      movel(p[0.462792, -0.058822, -0.000100, 0.000000, 3.141593, 0.000000],accel_mss,speed_ms,0,blend_radius_m)
      movel(p[0.463472, -0.058210, -0.000100, 0.000000, -3.141593, 0.000000],accel_mss,speed_ms,0,blend_radius_m)
      movel(p[0.463941, -0.057973, -0.000100, 0.000000, -3.141593, 0.000000],accel_mss,speed_ms,0,blend_radius_m)
      movel(p[0.464300, -0.058030, -0.000100, 0.000000, -3.141593, 0.000000],accel_mss,speed_ms,0,0.000)
      movel(p[0.464605, -0.058353, -0.000100, 0.000000, -3.141593, 0.000000],accel_mss,speed_ms,0,0.000)
      movel(p[0.464881, -0.058925, -0.000100, 0.000000, -3.141593, 0.000000],accel_mss,speed_ms,0,blend_radius_m)
      movel(p[0.465128, -0.059615, -0.000100, 0.000000, -3.141593, 0.000000],accel_mss,speed_ms,0,blend_radius_m)
      movel(p[0.465307, -0.060287, -0.000100, 0.000000, -3.141593, 0.000000],accel_mss,speed_ms,0,blend_radius_m)
      movel(p[0.465361, -0.060784, -0.000100, 0.000000, 3.141593, 0.000000],accel_mss,speed_ms,0,0.000)
      movel(p[0.465379, -0.061045, -0.000100, 0.000000, -3.141593, 0.000000],accel_mss,speed_ms,0,0.000)
      movel(p[0.465438, -0.061214, -0.000100, 0.000000, -3.141593, 0.000000],accel_mss,speed_ms,0,0.000)
      movel(p[0.465553, -0.061334, -0.000100, 0.000000, -3.141593, 0.000000],accel_mss,speed_ms,0,0.000)
      movel(p[0.465746, -0.061432, -0.000100, 0.000000, -3.141593, 0.000000],accel_mss,speed_ms,0,0.000)
      movel(p[0.466123, -0.061556, -0.000100, 0.000000, -3.141593, 0.000000],accel_mss,speed_ms,0,0.000)
      movel(p[0.466300, -0.061537, -0.000100, 0.000000, -3.141593, 0.000000],accel_mss,speed_ms,0,0.000)
      movel(p[0.466410, -0.061403, -0.000100, 0.000000, 3.141593, 0.000000],accel_mss,speed_ms,0,0.000)
      movel(p[0.466499, -0.061036, -0.000100, 0.000000, -3.141593, 0.000000],accel_mss,speed_ms,0,0.000)
      movel(p[0.466514, -0.060506, -0.000100, 0.000000, -3.141593, 0.000000],accel_mss,speed_ms,0,blend_radius_m)
      movel(p[0.466371, -0.059685, -0.000100, 0.000000, -3.141593, 0.000000],accel_mss,speed_ms,0,blend_radius_m)
      movel(p[0.466160, -0.058888, -0.000100, 0.000000, 3.141593, 0.000000],accel_mss,speed_ms,0,blend_radius_m)
      movel(p[0.465935, -0.058472, -0.000100, 0.000000, -3.141593, 0.000000],accel_mss,speed_ms,0,0.000)
      movel(p[0.465675, -0.058086, -0.000100, 0.000000, -3.141593, 0.000000],accel_mss,speed_ms,0,0.000)
      movel(p[0.465311, -0.057373, -0.000100, 0.000000, -3.141593, 0.000000],accel_mss,speed_ms,0,blend_radius_m)
      movel(p[0.464973, -0.056642, -0.000100, 0.000000, -3.141593, 0.000000],accel_mss,speed_ms,0,blend_radius_m)
      movel(p[0.464911, -0.056349, -0.000100, 0.000000, 3.141593, 0.000000],accel_mss,speed_ms,0,0.000)
      movel(p[0.464921, -0.056239, -0.000100, 0.000000, -3.141593, 0.000000],accel_mss,speed_ms,0,0.000)
      movel(p[0.464950, -0.056123, -0.000100, 0.000000, -3.141593, 0.000000],accel_mss,speed_ms,0,0.000)
      movel(p[0.464993, -0.056019, -0.000100, 0.000000, -3.141593, 0.000000],accel_mss,speed_ms,0,0.000)
      movel(p[0.465113, -0.055845, -0.000100, 0.000000, -3.141593, 0.000000],accel_mss,speed_ms,0,0.000)
      movel(p[0.465238, -0.055568, -0.000100, 0.000000, -3.141593, 0.000000],accel_mss,speed_ms,0,0.000)
      movel(p[0.465377, -0.055232, -0.000100, 0.000000, 3.141593, 0.000000],accel_mss,speed_ms,0,0.000)
      movel(p[0.465516, -0.054861, -0.000100, 0.000000, -3.141593, 0.000000],accel_mss,speed_ms,0,0.000)
      movel(p[0.465654, -0.054495, -0.000100, 0.000000, -3.141593, 0.000000],accel_mss,speed_ms,0,0.000)
      movel(p[0.465790, -0.054174, -0.000100, 0.000000, -3.141593, 0.000000],accel_mss,speed_ms,0,0.000)
      movel(p[0.465913, -0.053913, -0.000100, 0.000000, -3.141593, 0.000000],accel_mss,speed_ms,0,0.000)
      movel(p[0.466037, -0.053853, -0.000100, 0.000000, -3.141593, 0.000000],accel_mss,speed_ms,0,0.000)
      movel(p[0.466144, -0.053981, -0.000100, 0.000000, -3.141593, 0.000000],accel_mss,speed_ms,0,0.000)
      movel(p[0.466265, -0.054172, -0.000100, 0.000000, -3.141593, 0.000000],accel_mss,speed_ms,0,0.000)
      movel(p[0.466385, -0.054412, -0.000100, 0.000000, -3.141593, 0.000000],accel_mss,speed_ms,0,0.000)
      movel(p[0.466566, -0.054725, -0.000100, 0.000000, -3.141593, 0.000000],accel_mss,speed_ms,0,0.000)
      movel(p[0.466893, -0.055158, -0.000100, 0.000000, 3.141593, 0.000000],accel_mss,speed_ms,0,blend_radius_m)
      movel(p[0.467291, -0.055622, -0.000100, 0.000000, -3.141593, 0.000000],accel_mss,speed_ms,0,blend_radius_m)
      movel(p[0.467706, -0.056051, -0.000100, 0.000000, -3.141593, 0.000000],accel_mss,speed_ms,0,blend_radius_m)
      movel(p[0.468694, -0.056881, -0.000100, 0.000000, -3.141593, 0.000000],accel_mss,speed_ms,0,blend_radius_m)
      movel(p[0.469614, -0.057384, -0.000100, 0.000000, -3.141593, 0.000000],accel_mss,speed_ms,0,blend_radius_m)
      movel(p[0.470598, -0.057620, -0.000100, 0.000000, -3.141593, 0.000000],accel_mss,speed_ms,0,blend_radius_m)
      movel(p[0.471777, -0.057634, -0.000100, 0.000000, -3.141593, 0.000000],accel_mss,speed_ms,0,blend_radius_m)
      movel(p[0.473069, -0.057416, -0.000100, 0.000000, -3.141593, 0.000000],accel_mss,speed_ms,0,blend_radius_m)
      movel(p[0.474031, -0.056974, -0.000100, 0.000000, -3.141593, 0.000000],accel_mss,speed_ms,0,blend_radius_m)
      movel(p[0.474645, -0.056318, -0.000100, 0.000000, -3.141593, 0.000000],accel_mss,speed_ms,0,blend_radius_m)
      movel(p[0.474923, -0.055471, -0.000100, 0.000000, -3.141593, 0.000000],accel_mss,speed_ms,0,blend_radius_m)
      movel(p[0.474946, -0.055083, -0.000100, 0.000000, -3.141593, 0.000000],accel_mss,speed_ms,0,0.000)
      movel(p[0.474919, -0.054836, -0.000100, 0.000000, -3.141593, 0.000000],accel_mss,speed_ms,0,0.000)
      movel(p[0.474836, -0.054649, -0.000100, 0.000000, -3.141593, 0.000000],accel_mss,speed_ms,0,0.000)
      movel(p[0.474680, -0.054470, -0.000100, 0.000000, -3.141593, 0.000000],accel_mss,speed_ms,0,0.000)
      movel(p[0.474476, -0.054300, -0.000100, 0.000000, -3.141593, 0.000000],accel_mss,speed_ms,0,0.000)
      movel(p[0.474370, -0.054271, -0.000100, 0.000000, -3.141593, 0.000000],accel_mss,speed_ms,0,0.000)
      movel(p[0.474268, -0.054324, -0.000100, 0.000000, -3.141593, 0.000000],accel_mss,speed_ms,0,0.000)
      movel(p[0.474075, -0.054545, -0.000100, 0.000000, -3.141593, 0.000000],accel_mss,speed_ms,0,0.000)
      movel(p[0.473962, -0.054704, -0.000100, 0.000000, -3.141593, 0.000000],accel_mss,speed_ms,0,0.000)
      movel(p[0.473898, -0.054846, -0.000100, 0.000000, 3.141593, 0.000000],accel_mss,speed_ms,0,0.000)
      movel(p[0.473884, -0.054962, -0.000100, 0.000000, 3.141593, 0.000000],accel_mss,speed_ms,0,0.000)
      movel(p[0.473977, -0.055623, -0.000100, 0.000000, -3.141593, 0.000000],accel_mss,speed_ms,0,blend_radius_m)
      movel(p[0.473290, -0.056328, -0.000100, 0.000000, -3.141593, 0.000000],accel_mss,speed_ms,0,blend_radius_m)
      movel(p[0.472150, -0.056906, -0.000100, 0.000000, -3.141593, 0.000000],accel_mss,speed_ms,0,blend_radius_m)
      movel(p[0.470974, -0.057097, -0.000100, 0.000000, 3.141593, 0.000000],accel_mss,speed_ms,0,blend_radius_m)
      movel(p[0.470387, -0.057058, -0.000100, 0.000000, -3.141593, 0.000000],accel_mss,speed_ms,0,blend_radius_m)
      movel(p[0.469879, -0.056952, -0.000100, 0.000000, -3.141593, 0.000000],accel_mss,speed_ms,0,blend_radius_m)
      movel(p[0.469515, -0.056804, -0.000100, 0.000000, -3.141593, 0.000000],accel_mss,speed_ms,0,0.000)
      movel(p[0.469411, -0.056632, -0.000100, 0.000000, -3.141593, 0.000000],accel_mss,speed_ms,0,0.000)
      movel(p[0.469349, -0.056523, -0.000100, 0.000000, -3.141593, 0.000000],accel_mss,speed_ms,0,0.000)
      movel(p[0.469199, -0.056478, -0.000100, 0.000000, -3.141593, 0.000000],accel_mss,speed_ms,0,0.000)
      movel(p[0.468853, -0.056330, -0.000100, 0.000000, -3.141593, 0.000000],accel_mss,speed_ms,0,0.000)
      movel(p[0.467795, -0.055190, -0.000100, 0.000000, -3.141593, 0.000000],accel_mss,speed_ms,0,blend_radius_m)
      movel(p[0.466811, -0.054046, -0.000100, 0.000000, 3.141593, 0.000000],accel_mss,speed_ms,0,blend_radius_m)
      movel(p[0.466321, -0.053296, -0.000100, 0.000000, -3.141593, 0.000000],accel_mss,speed_ms,0,blend_radius_m)
      movel(p[0.466173, -0.052959, -0.000100, 0.000000, -3.141593, 0.000000],accel_mss,speed_ms,0,0.000)
      movel(p[0.466058, -0.052599, -0.000100, 0.000000, -3.141593, 0.000000],accel_mss,speed_ms,0,0.000)
      movel(p[0.465985, -0.052243, -0.000100, 0.000000, 3.141593, 0.000000],accel_mss,speed_ms,0,0.000)
      movel(p[0.465961, -0.051920, -0.000100, 0.000000, -3.141593, 0.000000],accel_mss,speed_ms,0,0.000)
      movel(p[0.465948, -0.051608, -0.000100, 0.000000, -3.141593, 0.000000],accel_mss,speed_ms,0,0.000)
      movel(p[0.465908, -0.051219, -0.000100, 0.000000, 3.141593, 0.000000],accel_mss,speed_ms,0,0.000)
      movel(p[0.465850, -0.050819, -0.000100, 0.000000, 3.141593, 0.000000],accel_mss,speed_ms,0,0.000)
      movel(p[0.465781, -0.050472, -0.000100, 0.000000, -3.141593, 0.000000],accel_mss,speed_ms,0,0.000)
      movel(p[0.465685, -0.050012, -0.000100, 0.000000, -3.141593, 0.000000],accel_mss,speed_ms,0,0.000)
      movel(p[0.465675, -0.049785, -0.000100, 0.000000, -3.141593, 0.000000],accel_mss,speed_ms,0,0.000)
      movel(p[0.465734, -0.049633, -0.000100, 0.000000, -3.141593, 0.000000],accel_mss,speed_ms,0,0.000)
      movel(p[0.465878, -0.049490, -0.000100, 0.000000, 3.141593, 0.000000],accel_mss,speed_ms,0,0.000)
      movel(p[0.465992, -0.049418, -0.000100, 0.000000, -3.141593, 0.000000],accel_mss,speed_ms,0,0.000)
      movel(p[0.466107, -0.049368, -0.000100, 0.000000, -3.141593, 0.000000],accel_mss,speed_ms,0,0.000)
      movel(p[0.466205, -0.049344, -0.000100, 0.000000, -3.141593, 0.000000],accel_mss,speed_ms,0,0.000)
      movel(p[0.466337, -0.049355, -0.000100, 0.000000, -3.141593, 0.000000],accel_mss,speed_ms,0,0.000)
      movel(p[0.466507, -0.049227, -0.000100, 0.000000, -3.141593, 0.000000],accel_mss,speed_ms,0,0.000)
      movel(p[0.466710, -0.049045, -0.000100, 0.000000, -3.141593, 0.000000],accel_mss,speed_ms,0,0.000)
      movel(p[0.466929, -0.048816, -0.000100, 0.000000, -3.141593, 0.000000],accel_mss,speed_ms,0,0.000)
      movel(p[0.467341, -0.048418, -0.000100, 0.000000, 3.141593, 0.000000],accel_mss,speed_ms,0,blend_radius_m)
      movel(p[0.467611, -0.048348, -0.000100, 0.000000, -3.141593, 0.000000],accel_mss,speed_ms,0,0.000)
      movel(p[0.467849, -0.048511, -0.000100, 0.000000, -3.141593, 0.000000],accel_mss,speed_ms,0,0.000)
      movel(p[0.468144, -0.049050, -0.000100, 0.000000, 3.141593, 0.000000],accel_mss,speed_ms,0,blend_radius_m)
      movel(p[0.468269, -0.049461, -0.000100, 0.000000, -3.141593, 0.000000],accel_mss,speed_ms,0,0.000)
      movel(p[0.468244, -0.049843, -0.000100, 0.000000, -3.141593, 0.000000],accel_mss,speed_ms,0,0.000)
      movel(p[0.468058, -0.050219, -0.000100, 0.000000, -3.141593, 0.000000],accel_mss,speed_ms,0,0.000)
      movel(p[0.467702, -0.050617, -0.000100, 0.000000, -3.141593, 0.000000],accel_mss,speed_ms,0,blend_radius_m)
      movel(p[0.467451, -0.050933, -0.000100, 0.000000, -3.141593, 0.000000],accel_mss,speed_ms,0,0.000)
      movel(p[0.467323, -0.051294, -0.000100, 0.000000, -3.141593, 0.000000],accel_mss,speed_ms,0,0.000)
      movel(p[0.467354, -0.051566, -0.000100, 0.000000, -3.141593, 0.000000],accel_mss,speed_ms,0,0.000)
      movel(p[0.467523, -0.051678, -0.000100, 0.000000, -3.141593, 0.000000],accel_mss,speed_ms,0,0.000)
      movel(p[0.467639, -0.051641, -0.000100, 0.000000, -3.141593, 0.000000],accel_mss,speed_ms,0,0.000)
      movel(p[0.467852, -0.051475, -0.000100, 0.000000, -3.141593, 0.000000],accel_mss,speed_ms,0,0.000)
      movel(p[0.468096, -0.051251, -0.000100, 0.000000, -3.141593, 0.000000],accel_mss,speed_ms,0,0.000)
      movel(p[0.468345, -0.050986, -0.000100, 0.000000, -3.141593, 0.000000],accel_mss,speed_ms,0,0.000)
      movel(p[0.468754, -0.050529, -0.000100, 0.000000, -3.141593, 0.000000],accel_mss,speed_ms,0,blend_radius_m)
      movel(p[0.468896, -0.050427, -0.000100, 0.000000, -3.141593, 0.000000],accel_mss,speed_ms,0,0.000)
      movel(p[0.468998, -0.050454, -0.000100, 0.000000, -3.141593, 0.000000],accel_mss,speed_ms,0,0.000)
      movel(p[0.469108, -0.050648, -0.000100, 0.000000, -3.141593, 0.000000],accel_mss,speed_ms,0,0.000)
      movel(p[0.469178, -0.050801, -0.000100, 0.000000, -3.141593, 0.000000],accel_mss,speed_ms,0,0.000)
      movel(p[0.469265, -0.050968, -0.000100, 0.000000, -3.141593, 0.000000],accel_mss,speed_ms,0,0.000)
      movel(p[0.469354, -0.051124, -0.000100, 0.000000, -3.141593, 0.000000],accel_mss,speed_ms,0,0.000)
      movel(p[0.469430, -0.051239, -0.000100, 0.000000, -3.141593, 0.000000],accel_mss,speed_ms,0,0.000)
      movel(p[0.469498, -0.051385, -0.000100, 0.000000, -3.141593, 0.000000],accel_mss,speed_ms,0,0.000)
      movel(p[0.469507, -0.051549, -0.000100, 0.000000, -3.141593, 0.000000],accel_mss,speed_ms,0,0.000)
      movel(p[0.469456, -0.051761, -0.000100, 0.000000, -3.141593, 0.000000],accel_mss,speed_ms,0,0.000)
      movel(p[0.469331, -0.052064, -0.000100, 0.000000, -3.141593, 0.000000],accel_mss,speed_ms,0,0.000)
      movel(p[0.469212, -0.052308, -0.000100, 0.000000, -3.141593, 0.000000],accel_mss,speed_ms,0,0.000)
      movel(p[0.469078, -0.052554, -0.000100, 0.000000, 3.141593, 0.000000],accel_mss,speed_ms,0,0.000)
      movel(p[0.468948, -0.052768, -0.000100, 0.000000, 3.141593, 0.000000],accel_mss,speed_ms,0,0.000)
      movel(p[0.468849, -0.052903, -0.000100, 0.000000, -3.141593, 0.000000],accel_mss,speed_ms,0,0.000)
      movel(p[0.468771, -0.053025, -0.000100, 0.000000, -3.141593, 0.000000],accel_mss,speed_ms,0,0.000)
      movel(p[0.468714, -0.053183, -0.000100, 0.000000, -3.141593, 0.000000],accel_mss,speed_ms,0,0.000)
      movel(p[0.468683, -0.053351, -0.000100, 0.000000, -3.141593, 0.000000],accel_mss,speed_ms,0,0.000)
      movel(p[0.468687, -0.053503, -0.000100, 0.000000, -3.141593, 0.000000],accel_mss,speed_ms,0,0.000)
      movel(p[0.468732, -0.053680, -0.000100, 0.000000, -3.141593, 0.000000],accel_mss,speed_ms,0,0.000)
      movel(p[0.468812, -0.053779, -0.000100, 0.000000, -3.141593, 0.000000],accel_mss,speed_ms,0,0.000)
      movel(p[0.468944, -0.053823, -0.000100, 0.000000, -3.141593, 0.000000],accel_mss,speed_ms,0,0.000)
      movel(p[0.469170, -0.053822, -0.000100, 0.000000, 3.141593, 0.000000],accel_mss,speed_ms,0,0.000)
      movel(p[0.469361, -0.053787, -0.000100, 0.000000, -3.141593, 0.000000],accel_mss,speed_ms,0,0.000)
      movel(p[0.469578, -0.053704, -0.000100, 0.000000, 3.141593, 0.000000],accel_mss,speed_ms,0,0.000)
      movel(p[0.469787, -0.053591, -0.000100, 0.000000, -3.141593, 0.000000],accel_mss,speed_ms,0,0.000)
      movel(p[0.469953, -0.053463, -0.000100, 0.000000, -3.141593, 0.000000],accel_mss,speed_ms,0,0.000)
      movel(p[0.470147, -0.053296, -0.000100, 0.000000, -3.141593, 0.000000],accel_mss,speed_ms,0,0.000)
      movel(p[0.470279, -0.053233, -0.000100, 0.000000, -3.141593, 0.000000],accel_mss,speed_ms,0,0.000)
      movel(p[0.470397, -0.053243, -0.000100, 0.000000, 3.141593, 0.000000],accel_mss,speed_ms,0,0.000)
      movel(p[0.470532, -0.053325, -0.000100, 0.000000, -3.141593, 0.000000],accel_mss,speed_ms,0,0.000)
      movel(p[0.470619, -0.053411, -0.000100, 0.000000, -3.141593, 0.000000],accel_mss,speed_ms,0,0.000)
      movel(p[0.470694, -0.053512, -0.000100, 0.000000, -3.141593, 0.000000],accel_mss,speed_ms,0,0.000)
      movel(p[0.470745, -0.053613, -0.000100, 0.000000, -3.141593, 0.000000],accel_mss,speed_ms,0,0.000)
      movel(p[0.470974, -0.054122, -0.000100, 0.000000, -3.141593, 0.000000],accel_mss,speed_ms,0,blend_radius_m)
      movel(p[0.471724, -0.054581, -0.000100, 0.000000, -3.141593, 0.000000],accel_mss,speed_ms,0,blend_radius_m)
      movel(p[0.472622, -0.054920, -0.000100, 0.000000, -3.141593, 0.000000],accel_mss,speed_ms,0,blend_radius_m)
      movel(p[0.473386, -0.054984, -0.000100, 0.000000, -3.141593, 0.000000],accel_mss,speed_ms,0,blend_radius_m)
      movel(p[0.473518, -0.054959, -0.000100, 0.000000, -3.141593, 0.000000],accel_mss,speed_ms,0,0.000)
      movel(p[0.473463, -0.054861, -0.000100, 0.000000, -3.141593, 0.000000],accel_mss,speed_ms,0,0.000)
      movel(p[0.473217, -0.054748, -0.000100, 0.000000, -3.141593, 0.000000],accel_mss,speed_ms,0,0.000)
      movel(p[0.473004, -0.054637, -0.000100, 0.000000, -3.141593, 0.000000],accel_mss,speed_ms,0,0.000)
      movel(p[0.472749, -0.054466, -0.000100, 0.000000, 3.141593, 0.000000],accel_mss,speed_ms,0,0.000)
      movel(p[0.472495, -0.054270, -0.000100, 0.000000, -3.141593, 0.000000],accel_mss,speed_ms,0,0.000)
      movel(p[0.472283, -0.054077, -0.000100, 0.000000, 3.141593, 0.000000],accel_mss,speed_ms,0,0.000)
      movel(p[0.471978, -0.053735, -0.000100, 0.000000, -3.141593, 0.000000],accel_mss,speed_ms,0,0.000)
      movel(p[0.471747, -0.053392, -0.000100, 0.000000, -3.141593, 0.000000],accel_mss,speed_ms,0,0.000)
      movel(p[0.471496, -0.052895, -0.000100, 0.000000, -3.141593, 0.000000],accel_mss,speed_ms,0,blend_radius_m)
      movel(p[0.471058, -0.051903, -0.000100, 0.000000, -3.141593, 0.000000],accel_mss,speed_ms,0,blend_radius_m)
      movel(p[0.470604, -0.050882, -0.000100, 0.000000, -3.141593, 0.000000],accel_mss,speed_ms,0,blend_radius_m)
      movel(p[0.470223, -0.050082, -0.000100, 0.000000, -3.141593, 0.000000],accel_mss,speed_ms,0,blend_radius_m)
      movel(p[0.469901, -0.049469, -0.000100, 0.000000, -3.141593, 0.000000],accel_mss,speed_ms,0,blend_radius_m)
      movel(p[0.469638, -0.049053, -0.000100, 0.000000, -3.141593, 0.000000],accel_mss,speed_ms,0,0.000)
      movel(p[0.469506, -0.048865, -0.000100, 0.000000, -3.141593, 0.000000],accel_mss,speed_ms,0,0.000)
      movel(p[0.469379, -0.048669, -0.000100, 0.000000, -3.141593, 0.000000],accel_mss,speed_ms,0,0.000)
      movel(p[0.469271, -0.048494, -0.000100, 0.000000, -3.141593, 0.000000],accel_mss,speed_ms,0,0.000)
      movel(p[0.469211, -0.048378, -0.000100, 0.000000, -3.141593, 0.000000],accel_mss,speed_ms,0,0.000)
      movel(p[0.469152, -0.048262, -0.000100, 0.000000, -3.141593, 0.000000],accel_mss,speed_ms,0,0.000)
      movel(p[0.469051, -0.048087, -0.000100, 0.000000, -3.141593, 0.000000],accel_mss,speed_ms,0,0.000)
      movel(p[0.468932, -0.047892, -0.000100, 0.000000, 3.141593, 0.000000],accel_mss,speed_ms,0,0.000)
      movel(p[0.468812, -0.047703, -0.000100, 0.000000, -3.141593, 0.000000],accel_mss,speed_ms,0,0.000)
      movel(p[0.468688, -0.047509, -0.000100, 0.000000, -3.141593, 0.000000],accel_mss,speed_ms,0,0.000)
      movel(p[0.468563, -0.047297, -0.000100, 0.000000, 3.141593, 0.000000],accel_mss,speed_ms,0,0.000)
      movel(p[0.468453, -0.047099, -0.000100, 0.000000, -3.141593, 0.000000],accel_mss,speed_ms,0,0.000)
      movel(p[0.468380, -0.046953, -0.000100, 0.000000, 3.141593, 0.000000],accel_mss,speed_ms,0,0.000)
      movel(p[0.468224, -0.046698, -0.000100, 0.000000, -3.141593, 0.000000],accel_mss,speed_ms,0,0.000)
      movel(p[0.467988, -0.046454, -0.000100, 0.000000, -3.141593, 0.000000],accel_mss,speed_ms,0,0.000)
      movel(p[0.467659, -0.046206, -0.000100, 0.000000, -3.141593, 0.000000],accel_mss,speed_ms,0,0.000)
      movel(p[0.467213, -0.045939, -0.000100, 0.000000, -3.141593, 0.000000],accel_mss,speed_ms,0,blend_radius_m)
      movel(p[0.466657, -0.045750, -0.000100, 0.000000, -3.141593, 0.000000],accel_mss,speed_ms,0,blend_radius_m)
      movel(p[0.465857, -0.045683, -0.000100, 0.000000, -3.141593, 0.000000],accel_mss,speed_ms,0,blend_radius_m)
      movel(p[0.464953, -0.045734, -0.000100, 0.000000, -3.141593, 0.000000],accel_mss,speed_ms,0,blend_radius_m)
      movel(p[0.464062, -0.045903, -0.000100, 0.000000, -3.141593, 0.000000],accel_mss,speed_ms,0,blend_radius_m)
      movel(p[0.463226, -0.046106, -0.000100, 0.000000, -3.141593, 0.000000],accel_mss,speed_ms,0,blend_radius_m)
      movel(p[0.462980, -0.046070, -0.000100, 0.000000, -3.141593, 0.000000],accel_mss,speed_ms,0,0.000)
      movel(p[0.462864, -0.045882, -0.000100, 0.000000, 3.141593, 0.000000],accel_mss,speed_ms,0,0.000)
      movel(p[0.462854, -0.045223, -0.000100, 0.000000, -3.141593, 0.000000],accel_mss,speed_ms,0,blend_radius_m)
      movel(p[0.462863, -0.044770, -0.000100, 0.000000, 3.141593, 0.000000],accel_mss,speed_ms,0,0.000)
      movel(p[0.462871, -0.044317, -0.000100, 0.000000, -3.141593, 0.000000],accel_mss,speed_ms,0,0.000)
      movel(p[0.462440, -0.043888, -0.000100, 0.000000, 3.141593, 0.000000],accel_mss,speed_ms,0,blend_radius_m)
      movel(p[0.462008, -0.043460, -0.000100, 0.000000, -3.141593, 0.000000],accel_mss,speed_ms,0,blend_radius_m)
      movel(p[0.461477, -0.042943, -0.000100, 0.000000, -3.141593, 0.000000],accel_mss,speed_ms,0,blend_radius_m)
      movel(p[0.461246, -0.042775, -0.000100, 0.000000, -3.141593, 0.000000],accel_mss,speed_ms,0,0.000)
      movel(p[0.461090, -0.042764, -0.000100, 0.000000, -3.141593, 0.000000],accel_mss,speed_ms,0,0.000)
      movel(p[0.460943, -0.042875, -0.000100, 0.000000, -3.141593, 0.000000],accel_mss,speed_ms,0,0.000)
      movel(p[0.460861, -0.043041, -0.000100, 0.000000, -3.141593, 0.000000],accel_mss,speed_ms,0,0.000)
      movel(p[0.460796, -0.043332, -0.000100, 0.000000, -3.141593, 0.000000],accel_mss,speed_ms,0,0.000)
      movel(p[0.460751, -0.043687, -0.000100, 0.000000, -3.141593, 0.000000],accel_mss,speed_ms,0,0.000)
      movel(p[0.460735, -0.044075, -0.000100, 0.000000, -3.141593, 0.000000],accel_mss,speed_ms,0,0.000)
      movel(p[0.460732, -0.044446, -0.000100, 0.000000, -3.141593, 0.000000],accel_mss,speed_ms,0,0.000)
      movel(p[0.460728, -0.044792, -0.000100, 0.000000, -3.141593, 0.000000],accel_mss,speed_ms,0,0.000)
      movel(p[0.460724, -0.045083, -0.000100, 0.000000, -3.141593, 0.000000],accel_mss,speed_ms,0,0.000)
      movel(p[0.460720, -0.045212, -0.000100, 0.000000, -3.141593, 0.000000],accel_mss,speed_ms,0,0.000)
      movel(p[0.460666, -0.045308, -0.000100, 0.000000, -3.141593, 0.000000],accel_mss,speed_ms,0,0.000)
      movel(p[0.460529, -0.045360, -0.000100, 0.000000, 3.141593, 0.000000],accel_mss,speed_ms,0,0.000)
      movel(p[0.460275, -0.045372, -0.000100, 0.000000, -3.141593, 0.000000],accel_mss,speed_ms,0,0.000)
      speed_ms    = 0.050
      movel(p[0.460275, -0.045372, 0.003000, 0.000000, -3.141593, 0.000000],accel_mss,speed_ms,0,blend_radius_m)
      speed_ms    = 1.000
      movel(p[0.460275, -0.045372, 0.015000, 0.000000, -3.141593, 0.000000],accel_mss,speed_ms,0,blend_radius_m)
      movel(p[0.386812, -0.046962, 0.015000, 0.000000, 3.141593, 0.000000],accel_mss,speed_ms,0,blend_radius_m)
      movel(p[0.386812, -0.046962, 0.003000, 0.000000, 3.141593, 0.000000],accel_mss,speed_ms,0,blend_radius_m)
      speed_ms    = 0.050
      movel(p[0.386812, -0.046962, -0.000100, 0.000000, 3.141593, 0.000000],accel_mss,speed_ms,0,blend_radius_m)
      speed_ms    = 0.083
      movel(p[0.386795, -0.048666, -0.000100, 0.000000, -3.141593, 0.000000],accel_mss,speed_ms,0,blend_radius_m)
      movel(p[0.386646, -0.050103, -0.000100, 0.000000, -3.141593, 0.000000],accel_mss,speed_ms,0,blend_radius_m)
      movel(p[0.386574, -0.050560, -0.000100, 0.000000, -3.141593, 0.000000],accel_mss,speed_ms,0,0.000)
      movel(p[0.386497, -0.051065, -0.000100, 0.000000, -3.141593, 0.000000],accel_mss,speed_ms,0,blend_radius_m)
      movel(p[0.386428, -0.051542, -0.000100, 0.000000, 3.141593, 0.000000],accel_mss,speed_ms,0,0.000)
      movel(p[0.386380, -0.051903, -0.000100, 0.000000, -3.141593, 0.000000],accel_mss,speed_ms,0,0.000)
      movel(p[0.386323, -0.052269, -0.000100, 0.000000, -3.141593, 0.000000],accel_mss,speed_ms,0,0.000)
      movel(p[0.386224, -0.052764, -0.000100, 0.000000, -3.141593, 0.000000],accel_mss,speed_ms,0,blend_radius_m)
      movel(p[0.386104, -0.053293, -0.000100, 0.000000, 3.141593, 0.000000],accel_mss,speed_ms,0,blend_radius_m)
      movel(p[0.385980, -0.053778, -0.000100, 0.000000, -3.141593, 0.000000],accel_mss,speed_ms,0,blend_radius_m)
      movel(p[0.385844, -0.054281, -0.000100, 0.000000, -3.141593, 0.000000],accel_mss,speed_ms,0,blend_radius_m)
      movel(p[0.385687, -0.054864, -0.000100, 0.000000, 3.141593, 0.000000],accel_mss,speed_ms,0,blend_radius_m)
      movel(p[0.385535, -0.055435, -0.000100, 0.000000, 3.141593, 0.000000],accel_mss,speed_ms,0,blend_radius_m)
      movel(p[0.385412, -0.055895, -0.000100, 0.000000, -3.141593, 0.000000],accel_mss,speed_ms,0,0.000)
      movel(p[0.385160, -0.056769, -0.000100, 0.000000, -3.141593, 0.000000],accel_mss,speed_ms,0,blend_radius_m)
      movel(p[0.384743, -0.058058, -0.000100, 0.000000, -3.141593, 0.000000],accel_mss,speed_ms,0,blend_radius_m)
      movel(p[0.384315, -0.059321, -0.000100, 0.000000, 3.141593, 0.000000],accel_mss,speed_ms,0,blend_radius_m)
      movel(p[0.384051, -0.060003, -0.000100, 0.000000, 3.141593, 0.000000],accel_mss,speed_ms,0,blend_radius_m)
      movel(p[0.383974, -0.060191, -0.000100, 0.000000, -3.141593, 0.000000],accel_mss,speed_ms,0,0.000)
      movel(p[0.383806, -0.060619, -0.000100, 0.000000, 3.141593, 0.000000],accel_mss,speed_ms,0,0.000)
      movel(p[0.383607, -0.061130, -0.000100, 0.000000, -3.141593, 0.000000],accel_mss,speed_ms,0,blend_radius_m)
      movel(p[0.383395, -0.061679, -0.000100, 0.000000, -3.141593, 0.000000],accel_mss,speed_ms,0,blend_radius_m)
      movel(p[0.383165, -0.062270, -0.000100, 0.000000, -3.141593, 0.000000],accel_mss,speed_ms,0,blend_radius_m)
      movel(p[0.382909, -0.062908, -0.000100, 0.000000, -3.141593, 0.000000],accel_mss,speed_ms,0,blend_radius_m)
      movel(p[0.382666, -0.063498, -0.000100, 0.000000, -3.141593, 0.000000],accel_mss,speed_ms,0,blend_radius_m)
      movel(p[0.382481, -0.063929, -0.000100, 0.000000, 3.141593, 0.000000],accel_mss,speed_ms,0,0.000)
      movel(p[0.382323, -0.064286, -0.000100, 0.000000, -3.141593, 0.000000],accel_mss,speed_ms,0,0.000)
      movel(p[0.382169, -0.064635, -0.000100, 0.000000, -3.141593, 0.000000],accel_mss,speed_ms,0,0.000)
      movel(p[0.382037, -0.064935, -0.000100, 0.000000, -3.141593, 0.000000],accel_mss,speed_ms,0,0.000)
      movel(p[0.381963, -0.065103, -0.000100, 0.000000, -3.141593, 0.000000],accel_mss,speed_ms,0,0.000)
      movel(p[0.381894, -0.065258, -0.000100, 0.000000, -3.141593, 0.000000],accel_mss,speed_ms,0,0.000)
      movel(p[0.381791, -0.065491, -0.000100, 0.000000, -3.141593, 0.000000],accel_mss,speed_ms,0,0.000)
      movel(p[0.381675, -0.065750, -0.000100, 0.000000, -3.141593, 0.000000],accel_mss,speed_ms,0,0.000)
      movel(p[0.381563, -0.066000, -0.000100, 0.000000, -3.141593, 0.000000],accel_mss,speed_ms,0,0.000)
      movel(p[0.381428, -0.066299, -0.000100, 0.000000, -3.141593, 0.000000],accel_mss,speed_ms,0,0.000)
      movel(p[0.381294, -0.066598, -0.000100, 0.000000, -3.141593, 0.000000],accel_mss,speed_ms,0,0.000)
      movel(p[0.381134, -0.065662, -0.000100, 0.000000, -3.141593, 0.000000],accel_mss,speed_ms,0,blend_radius_m)
      movel(p[0.380974, -0.064725, -0.000100, 0.000000, -3.141593, 0.000000],accel_mss,speed_ms,0,blend_radius_m)
      movel(p[0.380666, -0.063062, -0.000100, 0.000000, -3.141593, 0.000000],accel_mss,speed_ms,0,blend_radius_m)
      movel(p[0.380375, -0.061813, -0.000100, 0.000000, -3.141593, 0.000000],accel_mss,speed_ms,0,blend_radius_m)
      movel(p[0.380098, -0.060909, -0.000100, 0.000000, 3.141593, 0.000000],accel_mss,speed_ms,0,blend_radius_m)
      movel(p[0.379836, -0.060461, -0.000100, 0.000000, -3.141593, 0.000000],accel_mss,speed_ms,0,blend_radius_m)
      movel(p[0.379748, -0.060306, -0.000100, 0.000000, -3.141593, 0.000000],accel_mss,speed_ms,0,0.000)
      movel(p[0.379711, -0.060134, -0.000100, 0.000000, -3.141593, 0.000000],accel_mss,speed_ms,0,0.000)
      movel(p[0.379595, -0.059633, -0.000100, 0.000000, 3.141593, 0.000000],accel_mss,speed_ms,0,blend_radius_m)
      movel(p[0.378978, -0.058432, -0.000100, 0.000000, -3.141593, 0.000000],accel_mss,speed_ms,0,blend_radius_m)
      movel(p[0.378312, -0.057264, -0.000100, 0.000000, 3.141593, 0.000000],accel_mss,speed_ms,0,blend_radius_m)
      movel(p[0.377822, -0.056620, -0.000100, 0.000000, -3.141593, 0.000000],accel_mss,speed_ms,0,blend_radius_m)
      movel(p[0.377684, -0.056463, -0.000100, 0.000000, -3.141593, 0.000000],accel_mss,speed_ms,0,0.000)
      movel(p[0.377567, -0.056307, -0.000100, 0.000000, 3.141593, 0.000000],accel_mss,speed_ms,0,0.000)
      movel(p[0.377482, -0.056171, -0.000100, 0.000000, -3.141593, 0.000000],accel_mss,speed_ms,0,0.000)
      movel(p[0.377374, -0.055880, -0.000100, 0.000000, 3.141593, 0.000000],accel_mss,speed_ms,0,0.000)
      movel(p[0.375924, -0.054419, -0.000100, 0.000000, -3.141593, 0.000000],accel_mss,speed_ms,0,blend_radius_m)
      movel(p[0.374467, -0.052966, -0.000100, 0.000000, -3.141593, 0.000000],accel_mss,speed_ms,0,blend_radius_m)
      movel(p[0.374255, -0.052878, -0.000100, 0.000000, 3.141593, 0.000000],accel_mss,speed_ms,0,0.000)
      movel(p[0.373995, -0.052743, -0.000100, 0.000000, -3.141593, 0.000000],accel_mss,speed_ms,0,0.000)
      movel(p[0.373780, -0.052594, -0.000100, 0.000000, 3.141593, 0.000000],accel_mss,speed_ms,0,0.000)
      movel(p[0.373548, -0.052418, -0.000100, 0.000000, -3.141593, 0.000000],accel_mss,speed_ms,0,0.000)
      movel(p[0.372577, -0.051784, -0.000100, 0.000000, -3.141593, 0.000000],accel_mss,speed_ms,0,blend_radius_m)
      movel(p[0.371013, -0.051013, -0.000100, 0.000000, -3.141593, 0.000000],accel_mss,speed_ms,0,blend_radius_m)
      movel(p[0.369353, -0.050310, -0.000100, 0.000000, -3.141593, 0.000000],accel_mss,speed_ms,0,blend_radius_m)
      movel(p[0.368011, -0.049879, -0.000100, 0.000000, -3.141593, 0.000000],accel_mss,speed_ms,0,blend_radius_m)
      movel(p[0.366754, -0.049571, -0.000100, 0.000000, 3.141593, 0.000000],accel_mss,speed_ms,0,blend_radius_m)
      movel(p[0.365902, -0.049396, -0.000100, 0.000000, -3.141593, 0.000000],accel_mss,speed_ms,0,blend_radius_m)
      movel(p[0.365099, -0.049283, -0.000100, 0.000000, 3.141593, 0.000000],accel_mss,speed_ms,0,blend_radius_m)
      movel(p[0.364039, -0.049185, -0.000100, 0.000000, -3.141593, 0.000000],accel_mss,speed_ms,0,blend_radius_m)
      movel(p[0.363630, -0.049149, -0.000100, 0.000000, 3.141593, 0.000000],accel_mss,speed_ms,0,0.000)
      movel(p[0.363266, -0.049107, -0.000100, 0.000000, -3.141593, 0.000000],accel_mss,speed_ms,0,0.000)
      movel(p[0.362963, -0.049064, -0.000100, 0.000000, 3.141593, 0.000000],accel_mss,speed_ms,0,0.000)
      movel(p[0.362796, -0.048944, -0.000100, 0.000000, 3.141593, 0.000000],accel_mss,speed_ms,0,0.000)
      movel(p[0.362782, -0.048835, -0.000100, 0.000000, -3.141593, 0.000000],accel_mss,speed_ms,0,0.000)
      movel(p[0.362844, -0.048649, -0.000100, 0.000000, -3.141593, 0.000000],accel_mss,speed_ms,0,0.000)
      movel(p[0.363064, -0.048183, -0.000100, 0.000000, -3.141593, 0.000000],accel_mss,speed_ms,0,blend_radius_m)
      movel(p[0.363348, -0.047619, -0.000100, 0.000000, -3.141593, 0.000000],accel_mss,speed_ms,0,blend_radius_m)
      movel(p[0.363586, -0.047210, -0.000100, 0.000000, 3.141593, 0.000000],accel_mss,speed_ms,0,0.000)
      movel(p[0.363867, -0.046808, -0.000100, 0.000000, -3.141593, 0.000000],accel_mss,speed_ms,0,0.000)
      movel(p[0.364298, -0.046258, -0.000100, 0.000000, 3.141593, 0.000000],accel_mss,speed_ms,0,blend_radius_m)
      movel(p[0.364514, -0.045981, -0.000100, 0.000000, 3.141593, 0.000000],accel_mss,speed_ms,0,0.000)
      movel(p[0.364696, -0.045726, -0.000100, 0.000000, -3.141593, 0.000000],accel_mss,speed_ms,0,0.000)
      movel(p[0.364837, -0.045509, -0.000100, 0.000000, -3.141593, 0.000000],accel_mss,speed_ms,0,0.000)
      movel(p[0.364886, -0.045346, -0.000100, 0.000000, -3.141593, 0.000000],accel_mss,speed_ms,0,0.000)
      movel(p[0.365015, -0.045178, -0.000100, 0.000000, -3.141593, 0.000000],accel_mss,speed_ms,0,0.000)
      movel(p[0.365185, -0.044983, -0.000100, 0.000000, -3.141593, 0.000000],accel_mss,speed_ms,0,0.000)
      movel(p[0.365386, -0.044778, -0.000100, 0.000000, -3.141593, 0.000000],accel_mss,speed_ms,0,0.000)
      movel(p[0.365587, -0.044571, -0.000100, 0.000000, -3.141593, 0.000000],accel_mss,speed_ms,0,0.000)
      movel(p[0.365757, -0.044371, -0.000100, 0.000000, 3.141593, 0.000000],accel_mss,speed_ms,0,0.000)
      movel(p[0.365883, -0.044196, -0.000100, 0.000000, -3.141593, 0.000000],accel_mss,speed_ms,0,0.000)
      movel(p[0.365942, -0.044010, -0.000100, 0.000000, 3.141593, 0.000000],accel_mss,speed_ms,0,0.000)
      movel(p[0.366109, -0.043794, -0.000100, 0.000000, -3.141593, 0.000000],accel_mss,speed_ms,0,0.000)
      movel(p[0.366327, -0.043544, -0.000100, 0.000000, 3.141593, 0.000000],accel_mss,speed_ms,0,0.000)
      movel(p[0.366586, -0.043278, -0.000100, 0.000000, -3.141593, 0.000000],accel_mss,speed_ms,0,0.000)
      movel(p[0.366845, -0.043013, -0.000100, 0.000000, 3.141593, 0.000000],accel_mss,speed_ms,0,0.000)
      movel(p[0.367063, -0.042765, -0.000100, 0.000000, -3.141593, 0.000000],accel_mss,speed_ms,0,0.000)
      movel(p[0.367231, -0.042553, -0.000100, 0.000000, 3.141593, 0.000000],accel_mss,speed_ms,0,0.000)
      movel(p[0.367359, -0.042222, -0.000100, 0.000000, -3.141593, 0.000000],accel_mss,speed_ms,0,0.000)
      movel(p[0.368499, -0.041068, -0.000100, 0.000000, -3.141593, 0.000000],accel_mss,speed_ms,0,blend_radius_m)
      movel(p[0.369652, -0.039926, -0.000100, 0.000000, 3.141593, 0.000000],accel_mss,speed_ms,0,blend_radius_m)
      movel(p[0.369892, -0.039828, -0.000100, 0.000000, -3.141593, 0.000000],accel_mss,speed_ms,0,0.000)
      movel(p[0.370134, -0.039696, -0.000100, 0.000000, -3.141593, 0.000000],accel_mss,speed_ms,0,0.000)
      movel(p[0.370309, -0.039551, -0.000100, 0.000000, -3.141593, 0.000000],accel_mss,speed_ms,0,0.000)
      movel(p[0.370486, -0.039378, -0.000100, 0.000000, 3.141593, 0.000000],accel_mss,speed_ms,0,0.000)
      movel(p[0.370664, -0.039206, -0.000100, 0.000000, 3.141593, 0.000000],accel_mss,speed_ms,0,0.000)
      movel(p[0.370843, -0.039061, -0.000100, 0.000000, -3.141593, 0.000000],accel_mss,speed_ms,0,0.000)
      movel(p[0.371001, -0.038955, -0.000100, 0.000000, -3.141593, 0.000000],accel_mss,speed_ms,0,0.000)
      movel(p[0.371177, -0.038913, -0.000100, 0.000000, 3.141593, 0.000000],accel_mss,speed_ms,0,0.000)
      movel(p[0.371276, -0.038863, -0.000100, 0.000000, 3.141593, 0.000000],accel_mss,speed_ms,0,0.000)
      movel(p[0.371375, -0.038791, -0.000100, 0.000000, 3.141593, 0.000000],accel_mss,speed_ms,0,0.000)
      movel(p[0.371458, -0.038706, -0.000100, 0.000000, -3.141593, 0.000000],accel_mss,speed_ms,0,0.000)
      movel(p[0.371557, -0.038607, -0.000100, 0.000000, -3.141593, 0.000000],accel_mss,speed_ms,0,0.000)
      movel(p[0.371705, -0.038490, -0.000100, 0.000000, -3.141593, 0.000000],accel_mss,speed_ms,0,0.000)
      movel(p[0.371874, -0.038375, -0.000100, 0.000000, 3.141593, 0.000000],accel_mss,speed_ms,0,0.000)
      movel(p[0.372039, -0.038281, -0.000100, 0.000000, 3.141593, 0.000000],accel_mss,speed_ms,0,0.000)
      movel(p[0.372228, -0.038182, -0.000100, 0.000000, -3.141593, 0.000000],accel_mss,speed_ms,0,0.000)
      movel(p[0.372474, -0.038049, -0.000100, 0.000000, -3.141593, 0.000000],accel_mss,speed_ms,0,0.000)
      movel(p[0.372731, -0.037907, -0.000100, 0.000000, 3.141593, 0.000000],accel_mss,speed_ms,0,0.000)
      movel(p[0.372961, -0.037777, -0.000100, 0.000000, -3.141593, 0.000000],accel_mss,speed_ms,0,0.000)
      movel(p[0.373863, -0.037337, -0.000100, 0.000000, -3.141593, 0.000000],accel_mss,speed_ms,0,blend_radius_m)
      movel(p[0.374797, -0.037028, -0.000100, 0.000000, -3.141593, 0.000000],accel_mss,speed_ms,0,blend_radius_m)
      movel(p[0.375788, -0.036846, -0.000100, 0.000000, -3.141593, 0.000000],accel_mss,speed_ms,0,blend_radius_m)
      movel(p[0.376861, -0.036784, -0.000100, 0.000000, 3.141593, 0.000000],accel_mss,speed_ms,0,blend_radius_m)
      movel(p[0.378006, -0.036837, -0.000100, 0.000000, 3.141593, 0.000000],accel_mss,speed_ms,0,blend_radius_m)
      movel(p[0.379005, -0.037006, -0.000100, 0.000000, 3.141593, 0.000000],accel_mss,speed_ms,0,blend_radius_m)
      movel(p[0.379958, -0.037311, -0.000100, 0.000000, -3.141593, 0.000000],accel_mss,speed_ms,0,blend_radius_m)
      movel(p[0.380962, -0.037779, -0.000100, 0.000000, 3.141593, 0.000000],accel_mss,speed_ms,0,blend_radius_m)
      movel(p[0.381787, -0.038223, -0.000100, 0.000000, -3.141593, 0.000000],accel_mss,speed_ms,0,blend_radius_m)
      movel(p[0.382196, -0.038462, -0.000100, 0.000000, 3.141593, 0.000000],accel_mss,speed_ms,0,0.000)
      movel(p[0.382479, -0.038662, -0.000100, 0.000000, 3.141593, 0.000000],accel_mss,speed_ms,0,0.000)
      movel(p[0.382764, -0.038907, -0.000100, 0.000000, -3.141593, 0.000000],accel_mss,speed_ms,0,0.000)
      movel(p[0.382905, -0.039030, -0.000100, 0.000000, 3.141593, 0.000000],accel_mss,speed_ms,0,0.000)
      movel(p[0.383047, -0.039134, -0.000100, 0.000000, -3.141593, 0.000000],accel_mss,speed_ms,0,0.000)
      movel(p[0.383173, -0.039209, -0.000100, 0.000000, -3.141593, 0.000000],accel_mss,speed_ms,0,0.000)
      movel(p[0.383452, -0.039312, -0.000100, 0.000000, -3.141593, 0.000000],accel_mss,speed_ms,0,0.000)
      movel(p[0.384373, -0.040235, -0.000100, 0.000000, 3.141593, 0.000000],accel_mss,speed_ms,0,blend_radius_m)
      movel(p[0.385240, -0.041133, -0.000100, 0.000000, -3.141593, 0.000000],accel_mss,speed_ms,0,blend_radius_m)
      movel(p[0.385467, -0.041478, -0.000100, 0.000000, -3.141593, 0.000000],accel_mss,speed_ms,0,0.000)
      movel(p[0.385523, -0.041597, -0.000100, 0.000000, -3.141593, 0.000000],accel_mss,speed_ms,0,0.000)
      movel(p[0.385624, -0.041784, -0.000100, 0.000000, -3.141593, 0.000000],accel_mss,speed_ms,0,0.000)
      movel(p[0.385744, -0.041996, -0.000100, 0.000000, -3.141593, 0.000000],accel_mss,speed_ms,0,0.000)
      movel(p[0.385867, -0.042204, -0.000100, 0.000000, -3.141593, 0.000000],accel_mss,speed_ms,0,0.000)
      movel(p[0.386004, -0.042481, -0.000100, 0.000000, -3.141593, 0.000000],accel_mss,speed_ms,0,0.000)
      movel(p[0.386175, -0.042940, -0.000100, 0.000000, -3.141593, 0.000000],accel_mss,speed_ms,0,0.000)
      movel(p[0.386345, -0.043470, -0.000100, 0.000000, 3.141593, 0.000000],accel_mss,speed_ms,0,blend_radius_m)
      movel(p[0.386489, -0.044004, -0.000100, 0.000000, 3.141593, 0.000000],accel_mss,speed_ms,0,blend_radius_m)
      movel(p[0.386710, -0.045299, -0.000100, 0.000000, -3.141593, 0.000000],accel_mss,speed_ms,0,blend_radius_m)
      movel(p[0.386812, -0.046962, -0.000100, 0.000000, 3.141593, 0.000000],accel_mss,speed_ms,0,blend_radius_m)
      speed_ms    = 0.050
      movel(p[0.386812, -0.046962, 0.003000, 0.000000, 3.141593, 0.000000],accel_mss,speed_ms,0,blend_radius_m)
      speed_ms    = 1.000
      movel(p[0.386812, -0.046962, 0.015000, 0.000000, 3.141593, 0.000000],accel_mss,speed_ms,0,blend_radius_m)
      movel(p[0.516600, -0.149080, 0.015000, 0.000000, -3.141593, 0.000000],accel_mss,speed_ms,0,blend_radius_m)
      movel(p[0.516600, -0.149080, 0.045000, 0.000000, -3.141593, 0.000000],accel_mss,speed_ms,0,blend_radius_m)
      # End of main program
    end

    Machining1()
    $ 3 "Halt"
    halt
  end
end
